PROGRAM MAIN
VAR
	test2: BOOL;
	
	candle1	: ST_Candle;
	candle2	: ST_Candle;
	aCandles	: ARRAY[1..4, 1..4] OF ST_Candle;
	
END_VAR


Case_Chase();
gvl.timer1sec;

candle1.dia := 2.3;
candle1.height := 4;
aCandles;


candle1.weight := F_WeightCalc(dia:= candle1.dia, height:= candle1.height);

F_WeightCalcByReference(candle1);

END_PROGRAM

(* stored: Version 1.1.0.1, ProductVersion 3.1.4024.12
   POU MAIN: Id {cdbbbc71-3dd8-48a4-bcb5-7febaf611fb5}, SpecialFunc None *)
